{attribute 'qualified_only'}
VAR_GLOBAL
		
	ix_fotoCelTest : BOOL;
	qx_relaisTest : BOOL;
	
	// ingangen Noodstop
	ix_E_stopNC : BOOL;
	ix_E_stopNO : BOOL; 
	
	// ingangen fotocel
	ix_lengteFC : BOOL;
	ix_hamsterGripperDetectieFC : BOOL;
	
	ix_reedCuttingtoolCilinder : BOOL;
	ix_reedGripperCilinder1 : BOOL;
	ix_reedGripperCilinder2 : BOOL;
	
	// start/ stop uitgangen extruder&cutting tool
	qx_relaisExtruderStart : BOOL;
	qx_relaisExtruderStop: BOOL;
	qx_relaisCuttingtoolActiveer : BOOL;
	qx_relaisCuttingtoolDeactiveer : BOOL;
	
	//uitgangen gereserveerd voor KUKA/Engel communicatie
	// E stop
	// bitlevel comm's
	qx_kukaCommEstop : BOOL; // E_stop
	qx_kukaComm2 : BOOL; // sein veilig
	qx_kukaComm3 : BOOL; // startcommando
	qx_kukaComm4 : BOOL; // alarm
	qx_kukaComm5 : BOOL; // ander spul weet ik veel
	
END_VAR

(* stored: Version 1.1.0.1, ProductVersion 3.1.4024.12
   GVL DB10_Alias: Id {125f7c14-bc07-4185-8080-6bf9d7d4c446} *)
